(* PLC project Traffic control simulator, CODESYS CODESYS V3.5 SP16, author Toni Kucic *)
(* stored: creationDateTime 2021-03-25T19:26:30.1030266, version 1.0, modificationDateTime 2021-03-25T19:26:13.0193121, organization TK Automation *)
(* Traffic control is often used a simple introduction into sequencing when programming PLCs. As a part of my portfolio I have written a simple timing controller and a simulator for two crossroads that are one way streets with pedestrians going in all directions. The project is meant for begginers and for educational purposes. It is published under MIT license. Written in CODESYS 3.5 and in structured text language. *)

TYPE SpriteDef_typ : STRUCT
  x : INT;  (* Initial position of the sprite *)
  y : INT;  (* Initial position of the sprite *)
  speed : INT;  (* Initial speed of the sprite *)
  width : INT;  (* Sprites width *)
  height : INT;  (* Sprites height *)
  screenWidth : INT;  (* Screen width *)
  screenHeight : INT;  (* Screen height *)
END_STRUCT;
END_TYPE

TYPE trafficLightCars : STRUCT
  RedLamp : BOOL;  (* TRUE: Red lamp is on *)
  YellowLamp : BOOL;  (* TRUE: Yellow lamp is on *)
  GreenLamp : BOOL;  (* TRUE: Green lamp is on *)
END_STRUCT;
END_TYPE

TYPE trafficLightPed : STRUCT
  RedLight : BOOL;  (* TRUE: Red lamp is on *)
  GreenLight : BOOL;  (* TRUE: Green lamp is on *)
  TimeToSequenceChange : UINT;  (* Time in seconds until next light change *)
END_STRUCT;
END_TYPE

FUNCTION isSpriteColliding : BOOL
  VAR_INPUT
    sprite1 : Sprite;  (* Sprite 1 function block *)
    sprite2 : Sprite;  (* Sprite 2 function block *)
  END_VAR

            (*Calculate if these two sprites are overlapping*)
IF sprite1.actX < (sprite2.actX + sprite2.init.width) AND
   (sprite1.actX + sprite1.init.width) > sprite2.actX AND
   sprite1.actY < (sprite2.actY + sprite2.init.height) AND
  ( sprite1.init.height + sprite1.actY) > sprite2.actY THEN
   isSpriteColliding := TRUE;
ELSE
	isSpriteColliding := FALSE;
END_IF
          
END_FUNCTION

FUNCTION_BLOCK Sprite
  VAR_INPUT
    init : SpriteDef_typ;  (* Sprite initialization pars *)
    goTo : ARRAY[0..1] OF INT;  (* Sprite moves to x,y destination *)
    moveX : INT;  (* Moves the sprite by given ammount on the X axis *)
    moveY : INT;  (* Moves the sprite by given ammount on the Y axis *)
  END_VAR
  VAR_OUTPUT
    x : INT;  (* X position of the sprite *)
    y : INT;  (* Y position of the sprite *)
    atDestination : BOOL;  (* Flag to say it has arrived at its destination *)
    actX : INT;  (* Actual position on the screen, X axis *)
    actY : INT;  (* Actual position on the screen, Y axis *)
  END_VAR
  VAR
    vInit : BOOL := TRUE;  (* Initialization flag *)
    vSpriteDef : SpriteDef_typ;  (* Used sprite definition *)
    vActualX : INT;  (* Actual position on the screen, X axis *)
    vActualY : INT;  (* Actual position on the screen, Y axis *)
  END_VAR

            (*Initialize sprite on first scan*)
IF vInit THEN
	vSpriteDef := init;
	vInit := FALSE;
END_IF

(* Actual moving of the coordinates *)
vSpriteDef.x := vSpriteDef.x + moveX;
vSpriteDef.y := vSpriteDef.y + moveY;

(* Reseting the position if sprite goes off screen *)
(* If moving left to right *)
IF vSpriteDef.x > vSpriteDef.screenWidth THEN
	vSpriteDef.x := -vSpriteDef.width;
(* If moving right to left *)
ELSIF vSpriteDef.x < -vSpriteDef.width THEN
	vSpriteDef.x := vSpriteDef.screenWidth;	
END_IF
(* If moving from up, down *)
IF vSpriteDef.y > vSpriteDef.screenHeight THEN
	vSpriteDef.y := -vSpriteDef.height;
(* If moving from down, up *)
ELSIF vSpriteDef.y < -vSpriteDef.height THEN
	vSpriteDef.y := vSpriteDef.screenHeight;	
END_IF

(*x, y will be used to connect to absoulte movements of the graphic element*)
x := vSpriteDef.x - init.x;
y := vSpriteDef.y - init.y;

(*ActX and ActY will be used in the logic for e.g. object collision detection*)
actX := vSpriteDef.x;
actY := vSpriteDef.y;
          
END_FUNCTION_BLOCK

PROGRAM simulator
  VAR
    carC1HR : Sprite := (init := (screenHeight := 720, screenWidth := 1980, height := 80, width := 200, x := 568, y := 264));  (* Sprite controling car C1HR *)
    carC1HL : Sprite := (init := (screenHeight := 720, screenWidth := 1980, height := 80, width := 200, x := -50, y := 370));  (* Sprite controling car C1HL *)
    carC1VU : Sprite := (init := (screenHeight := 720, screenWidth := 1980, height := 200, width := 80, x := 270, y := -50));  (* Sprite controling car C1VU *)
    carC1VD : Sprite := (init := (screenHeight := 720, screenWidth := 1980, height := 200, width := 80, x := 372, y := 565));  (* Sprite controling car C1VD *)
    carC2VU : Sprite := (init := (screenHeight := 720, screenWidth := 1980, height := 200, width := 80, x := 1528, y := -50));  (* Sprite controling car C2VU *)
    carC2VD : Sprite := (init := (screenHeight := 720, screenWidth := 1980, height := 200, width := 80, x := 1631, y := 580));  (* Sprite controling car C2VD *)
    pedC1VU : Sprite := (init := (screenHeight := 720, screenWidth := 1980, height := 50, width := 50, x := 171, y := 7));  (* Sprite controling pedestrian C1VU *)
    pedC1VD : Sprite := (init := (screenHeight := 720, screenWidth := 1980, height := 50, width := 50, x := 486, y := 657));  (* Sprite controling pedestrian C1VD *)
    pedC2VU : Sprite := (init := (screenHeight := 720, screenWidth := 1980, height := 50, width := 50, x := 1427, y := 2));  (* Sprite controling pedestrian C2VU *)
    pedC2VD : Sprite := (init := (screenHeight := 720, screenWidth := 1980, height := 50, width := 50, x := 1742, y := 654));  (* Sprite controling pedestrian C2VD *)
    pedC1HL : Sprite := (init := (screenHeight := 720, screenWidth := 1980, height := 50, width := 50, x := 9, y := 491));  (* Sprite controling pedestrian C1HL *)
    pedC2HR : Sprite := (init := (screenHeight := 720, screenWidth := 1980, height := 50, width := 50, x := 1916, y := 174));  (* Sprite controling pedestrian C1HR *)
    Cross1CarU : trafficLightCars;  (* Car traffic light - Crossroad 1 - Cars going up to down *)
    Cross1CarD : trafficLightCars;  (* Car traffic light - Crossroad 1 - Cars going down to up *)
    Cross1CarL : trafficLightCars;  (* Car traffic light - Crossroad 1 - Cars going left to right *)
    Cross1CarR : trafficLightCars;  (* Car traffic light - Crossroad 1 - Cars going right to left *)
    Cross2CarU : trafficLightCars;  (* Car light - Crossroad 2 - Cars going up to down *)
    Cross2CarD : trafficLightCars;  (* Car light - Crossroad 2 - Cars going down to up *)
    Cross2CarL : trafficLightCars;  (* Car light - Crossroad 2 - Cars going left to right *)
    Cross2CarR : trafficLightCars;  (* Car light - Crossroad 2 - Cars going right to left *)
    Cross1PedLUD : trafficLightPed;  (* Pedestrian light - Crossroad 1 - Pedestrians going up to down on left side *)
    Cross1PedLDU : trafficLightPed;  (* Pedestrian light - Crossroad 1 - Pedestrians going down to up on left side *)
    Cross1PedRUD : trafficLightPed;  (* Pedestrian light - Crossroad 1 - Pedestrians going up to down on right side *)
    Cross1PedRDU : trafficLightPed;  (* Pedestrian light - Crossroad 1 - Pedestrians going down to up on right side *)
    Cross1PedULR : trafficLightPed;  (* Pedestrian light - Crossroad 1 - Pedestrians going left to right on upper side *)
    Cross1PedURL : trafficLightPed;  (* Pedestrian light - Crossroad 1 - Pedestrians going right to left on upper side *)
    Cross1PedDLR : trafficLightPed;  (* Pedestrian light - Crossroad 1 - Pedestrians going left to right on lower side *)
    Cross1PedDRL : trafficLightPed;  (* Pedestrian light - Crossroad 1 - Pedestrians going right to left on lower side *)
    Cross2PedLUD : trafficLightPed;  (* Pedestrian light - Crossroad 2 - Pedestrians going up to down on left side *)
    Cross2PedLDU : trafficLightPed;  (* Pedestrian light - Crossroad 2 - Pedestrians going down to up on left side *)
    Cross2PedRUD : trafficLightPed;  (* Pedestrian light - Crossroad 2 - Pedestrians going up to down on right side *)
    Cross2PedRDU : trafficLightPed;  (* Pedestrian light - Crossroad 2 - Pedestrians going down to up on right side *)
    Cross2PedULR : trafficLightPed;  (* Pedestrian light - Crossroad 2 - Pedestrians going left to right on upper side *)
    Cross2PedURL : trafficLightPed;  (* Pedestrian light - Crossroad 2 - Pedestrians going right to left on upper side *)
    Cross2PedDLR : trafficLightPed;  (* Pedestrian light - Crossroad 2 - Pedestrians going left to right on lower side *)
    Cross2PedDRL : trafficLightPed;  (* Pedestrian light - Crossroad 2 - Pedestrians going right to left on lower side *)
    vCollision : BOOL;  (* Collission has occured *)
    vDangerousCombination : BOOL;  (* Dangerous combination of lights has been detected *)
    vPoliceControl : BOOL;  (* Police control activated *)
    vCrashFlagX : INT := -200;  (* If collission is detected, holds position of collission x axis *)
    vCrashFlagY : INT := -200;  (* If collission is detected, holds position of collission y axis *)
    Blinker : BLINK;  (* Code that blinks a variable *)
    vFaultReason : STRING(255);  (* If collission or dangerous combination detected, holds more information where it has occured *)
  END_VAR

                    MOVE_CARS();
MOVE_PEDESTRIANS();

(*Blink yellow signal if the police is under control*)
IF vPoliceControl THEN
	UPDATE_OBJECTS();
	BLINK_YELLOW_SIGNAL();
(*Freeze situation if a collission or dangerous situation has occured*)
ELSIF vCollision OR vDangerousCombination THEN
	BLINK_DANGER_SIGNAL();
ELSE
	(*Everything is fine so move objects and let the main control the lights*)
	UPDATE_OBJECTS();
	CONTROL_LIGHTS();
	vFaultReason := '';
END_IF
FAULT_MONITOR();
gIO.PoliceModeActivated := vPoliceControl;
Blinker(ENABLE:=TRUE, TIMELOW:=T#1S, TIMEHIGH:=T#1S);



                  

ACTION CHECK_COLLISSIONS:
                        (*Check for collisions between each car with another car and pedestrian*)
vCollision := FALSE;

(*Collission car -> car*)
IF isSpriteColliding(carC1HR, carC1HL) THEN
	vCollision := TRUE;
	vCrashFlagX := carC1HR.actX;
	vCrashFlagY := carC1HL.actY;
	vFaultReason := 'COLLISSION AT CAR C1HR AND CAR C1HL';
END_IF
IF isSpriteColliding(carC1HR, carC1VU) THEN
	vCollision := TRUE;
	vCrashFlagX := carC1HR.actX;
	vCrashFlagY := carC1VU.actY;
	vFaultReason := 'COLLISSION AT CAR C1HR AND CAR C1VU';
END_IF
IF isSpriteColliding(carC1HR, carC1VD) THEN
	vCollision := TRUE;
	vCrashFlagX := carC1HR.actX;
	vCrashFlagY := carC1VD.actY;
	vFaultReason := 'COLLISSION AT CAR C1HR AND CAR C1VD';
END_IF
IF isSpriteColliding(carC1HR, carC2VD) THEN
	vCollision := TRUE;
	vCrashFlagX := carC1HR.actX;
	vCrashFlagY := carC2VD.actY;
	vFaultReason := 'COLLISSION AT CAR C1HR AND CAR C2VD';
END_IF
IF isSpriteColliding(carC1HR, carC2VU) THEN
	vCollision := TRUE;
	vCrashFlagX := carC1HR.actX;
	vCrashFlagY := carC2VU.actY;
	vFaultReason := 'COLLISSION AT CAR C1HR AND CAR C2VU';
END_IF
IF isSpriteColliding(carC1HL, carC1VU) THEN
	vCollision := TRUE;
	vCrashFlagX := carC1HL.actX;
	vCrashFlagY := carC1VU.actY;
	vFaultReason := 'COLLISSION AT CAR C1HL AND CAR C1VU';
END_IF
IF isSpriteColliding(carC1HL, carC1VD) THEN
	vCollision := TRUE;
	vCrashFlagX := carC1HL.actX;
	vCrashFlagY := carC1VD.actY;
	vFaultReason := 'COLLISSION AT CAR C1HL AND CAR C1VD';
END_IF
IF isSpriteColliding(carC1HL, carC2VU) THEN
	vCollision := TRUE;
	vCrashFlagX := carC1HL.actX;
	vCrashFlagY := carC2VU.actY;
	vFaultReason := 'COLLISSION AT CAR C1HL AND CAR C2VU';
END_IF
IF isSpriteColliding(carC1HL, carC2VD) THEN
	vCollision := TRUE;
	vCrashFlagX := carC1HL.actX;
	vCrashFlagY := carC2VD.actY;
	vFaultReason := 'COLLISSION AT CAR C1HL AND CAR C2VD';
END_IF
IF isSpriteColliding(carC1VU, carC1VD) THEN
	vCollision := TRUE;
	vCrashFlagX := carC1VU.actX;
	vCrashFlagY := carC1VD.actY;
	vFaultReason := 'COLLISSION AT CAR C1VU AND CAR C1VD';
END_IF
IF isSpriteColliding(carC1VU, carC2VD) THEN
	vCollision := TRUE;
	vCrashFlagX := carC1VU.actX;
	vCrashFlagY := carC2VD.actY;
	vFaultReason := 'COLLISSION AT CAR C1VU AND CAR C2VD';
END_IF
IF isSpriteColliding(carC1VU, carC2VU) THEN
	vCollision := TRUE;
	vCrashFlagX := carC1VU.actX;
	vCrashFlagY := carC2VU.actY;
	vFaultReason := 'COLLISSION AT CAR C1VU AND CAR C2VU';
END_IF
IF isSpriteColliding(carC1VD, carC2VD) THEN
	vCollision := TRUE;
	vCrashFlagX := carC1VD.actX;
	vCrashFlagY := carC2VD.actY;
	vFaultReason := 'COLLISSION AT CAR C1VD AND CAR C2VD';
END_IF
IF isSpriteColliding(carC1VD, carC2VU) THEN
	vCollision := TRUE; 
	vCrashFlagX := carC1VD.actX;
	vCrashFlagY := carC2VU.actY;
	vFaultReason := 'COLLISSION AT CAR C1VD AND CAR C2VU';
END_IF
IF isSpriteColliding(carC2VD, carC2VU) THEN
	vCollision := TRUE; 
	vCrashFlagX := carC2VD.actX;
	vCrashFlagY := carC2VU.actY;
	vFaultReason := 'COLLISSION AT CAR C2VD AND CAR C2VU';
END_IF

(*Check collission car -> pedestrian*)
IF isSpriteColliding(carC1HR, pedC1HL) THEN
	vCollision := TRUE;
	vCrashFlagX := carC1HR.actX;
	vCrashFlagY := pedC1HL.actY;
	vFaultReason := 'COLLISSION AT CAR C1HR AND PEDESTRIAN C1HL';
END_IF
IF isSpriteColliding(carC1HR, pedC1VU) THEN
	vCollision := TRUE;
	vCrashFlagX := carC1HR.actX;
	vCrashFlagY := pedC1VU.actY;
	vFaultReason := 'COLLISSION AT CAR C1HR AND PEDESTRIAN C1VU';
END_IF
IF isSpriteColliding(carC1HR, pedC1VD) THEN
	vCollision := TRUE;
	vCrashFlagX := carC1HR.actX;
	vCrashFlagY := pedC1VD.actY;
	vFaultReason := 'COLLISSION AT CAR C1HR AND PEDESTRIAN C1VD';
END_IF
IF isSpriteColliding(carC1HR, pedC2VU) THEN
	vCollision := TRUE;
	vCrashFlagX := carC1HR.actX;
	vCrashFlagY := pedC2VU.actY;
	vFaultReason := 'COLLISSION AT CAR C1HR AND PEDESTRIAN C2VU';
END_IF
IF isSpriteColliding(carC1HR, pedC2VD) THEN
	vCollision := TRUE;
	vCrashFlagX := carC1HR.actX;
	vCrashFlagY := pedC2VD.actY;
	vFaultReason := 'COLLISSION AT CAR C1HR AND PEDESTRIAN C2VD';
END_IF
IF isSpriteColliding(carC1HR, pedC2HR) THEN
	vCollision := TRUE;
	vCrashFlagX := carC1HR.actX;
	vCrashFlagY := pedC2HR.actY;
	vFaultReason := 'COLLISSION AT CAR C1HR AND PEDESTRIAN C2HR';
END_IF


IF isSpriteColliding(carC1HL, pedC1HL) THEN
	vCollision := TRUE;
	vCrashFlagX := carC1HL.actX;
	vCrashFlagY := pedC1HL.actY;
	vFaultReason := 'COLLISSION AT CAR C1HL AND PEDESTRIAN C1HL';
END_IF
IF isSpriteColliding(carC1HL, pedC1VU) THEN
	vCollision := TRUE;
	vCrashFlagX := carC1HL.actX;
	vCrashFlagY := pedC1VU.actY;
	vFaultReason := 'COLLISSION AT CAR C1HL AND PEDESTRIAN C1VU';
END_IF
IF isSpriteColliding(carC1HL, pedC1VD) THEN
	vCollision := TRUE;
	vCrashFlagX := carC1HL.actX;
	vCrashFlagY := pedC1VD.actY;
	vFaultReason := 'COLLISSION AT CAR C1HL AND PEDESTRIAN C1VD';
END_IF
IF isSpriteColliding(carC1HL, pedC2VU) THEN
	vCollision := TRUE;
	vCrashFlagX := carC1HL.actX;
	vCrashFlagY := pedC2VU.actY;
	vFaultReason := 'COLLISSION AT CAR C1HL AND PEDESTRIAN C2VU';
END_IF
IF isSpriteColliding(carC1HL, pedC2VD) THEN
	vCollision := TRUE;
	vCrashFlagX := carC1HL.actX;
	vCrashFlagY := pedC2VD.actY;
	vFaultReason := 'COLLISSION AT CAR C1HL AND PEDESTRIAN C2VD';
END_IF
IF isSpriteColliding(carC1HL, pedC2HR) THEN
	vCollision := TRUE;
	vCrashFlagX := carC1HL.actX;
	vCrashFlagY := pedC2HR.actY;
	vFaultReason := 'COLLISSION AT CAR C1HL AND PEDESTRIAN C2HR';
END_IF


IF isSpriteColliding(carC1VU, pedC1HL) THEN
	vCollision := TRUE;
	vCrashFlagX := carC1VU.actX;
	vCrashFlagY := pedC1HL.actY;
	vFaultReason := 'COLLISSION AT CAR C1VU AND PEDESTRIAN C1HL';
END_IF
IF isSpriteColliding(carC1VU, pedC1VU) THEN
	vCollision := TRUE;
	vCrashFlagX := carC1VU.actX;
	vCrashFlagY := pedC1VU.actY;
	vFaultReason := 'COLLISSION AT CAR C1VU AND PEDESTRIAN C1VU';
END_IF
IF isSpriteColliding(carC1VU, pedC1VD) THEN
	vCollision := TRUE;
	vCrashFlagX := carC1VU.actX;
	vCrashFlagY := pedC1VD.actY;
	vFaultReason := 'COLLISSION AT CAR C1VU AND PEDESTRIAN C1VD';
END_IF
IF isSpriteColliding(carC1VU, pedC2VU) THEN
	vCollision := TRUE;
	vCrashFlagX := carC1VU.actX;
	vCrashFlagY := pedC2VU.actY;
	vFaultReason := 'COLLISSION AT CAR C1VU AND PEDESTRIAN C2VU';
END_IF
IF isSpriteColliding(carC1VU, pedC2VD) THEN
	vCollision := TRUE;
	vCrashFlagX := carC1VU.actX;
	vCrashFlagY := pedC2VD.actY;
	vFaultReason := 'COLLISSION AT CAR C1VU AND PEDESTRIAN C2VD';
END_IF
IF isSpriteColliding(carC1VU, pedC2HR) THEN
	vCollision := TRUE;
	vCrashFlagX := carC1VU.actX;
	vCrashFlagY := pedC2HR.actY;
	vFaultReason := 'COLLISSION AT CAR C1VU AND PEDESTRIAN C2HR';
END_IF


IF isSpriteColliding(carC1VD, pedC1HL) THEN
	vCollision := TRUE;
	vCrashFlagX := carC1VD.actX;
	vCrashFlagY := pedC1HL.actY;
	vFaultReason := 'COLLISSION AT CAR C1VD AND PEDESTRIAN C1HL';
END_IF
IF isSpriteColliding(carC1VD, pedC1VU) THEN
	vCollision := TRUE;
	vCrashFlagX := carC1VD.actX;
	vCrashFlagY := pedC1VU.actY;
	vFaultReason := 'COLLISSION AT CAR C1VD AND PEDESTRIAN C1VU';
END_IF
IF isSpriteColliding(carC1VD, pedC1VD) THEN
	vCollision := TRUE;
	vCrashFlagX := carC1VD.actX;
	vCrashFlagY := pedC1VD.actY;
	vFaultReason := 'COLLISSION AT CAR C1VD AND PEDESTRIAN C1VD';
END_IF
IF isSpriteColliding(carC1VD, pedC2VU) THEN
	vCollision := TRUE;
	vCrashFlagX := carC1VD.actX;
	vCrashFlagY := pedC2VU.actY;
	vFaultReason := 'COLLISSION AT CAR C1VD AND PEDESTRIAN C2VU';
END_IF
IF isSpriteColliding(carC1VD, pedC2VD) THEN
	vCollision := TRUE;
	vCrashFlagX := carC1VD.actX;
	vCrashFlagY := pedC2VD.actY;
	vFaultReason := 'COLLISSION AT CAR C1VD AND PEDESTRIAN C2VD';
END_IF
IF isSpriteColliding(carC1VD, pedC2HR) THEN
	vCollision := TRUE;
	vCrashFlagX := carC1VD.actX;
	vCrashFlagY := pedC2HR.actY;
	vFaultReason := 'COLLISSION AT CAR C1VD AND PEDESTRIAN C2HR';
END_IF


IF isSpriteColliding(carC2VU, pedC1HL) THEN
	vCollision := TRUE;
	vCrashFlagX := carC2VU.actX;
	vCrashFlagY := pedC1HL.actY;
	vFaultReason := 'COLLISSION AT CAR C2VU AND PEDESTRIAN C1HL';
END_IF
IF isSpriteColliding(carC2VU, pedC1VU) THEN
	vCollision := TRUE;
	vCrashFlagX := carC2VU.actX;
	vCrashFlagY := pedC1VU.actY;
	vFaultReason := 'COLLISSION AT CAR C2VU AND PEDESTRIAN C1VU';
END_IF
IF isSpriteColliding(carC2VU, pedC1VD) THEN
	vCollision := TRUE;
	vCrashFlagX := carC2VU.actX;
	vCrashFlagY := pedC1VD.actY;
	vFaultReason := 'COLLISSION AT CAR C2VU AND PEDESTRIAN C1VD';
END_IF
IF isSpriteColliding(carC2VU, pedC2VU) THEN
	vCollision := TRUE;
	vCrashFlagX := carC2VU.actX;
	vCrashFlagY := pedC2VU.actY;
	vFaultReason := 'COLLISSION AT CAR C2VU AND PEDESTRIAN C2VU';
END_IF
IF isSpriteColliding(carC2VU, pedC2VD) THEN
	vCollision := TRUE;
	vCrashFlagX := carC2VU.actX;
	vCrashFlagY := pedC2VD.actY;
	vFaultReason := 'COLLISSION AT CAR C2VU AND PEDESTRIAN C2VD';
END_IF
IF isSpriteColliding(carC2VU, pedC2HR) THEN
	vCollision := TRUE;
	vCrashFlagX := carC2VU.actX;
	vCrashFlagY := pedC2HR.actY;
	vFaultReason := 'COLLISSION AT CAR C2VU AND PEDESTRIAN C2HR';
END_IF


IF isSpriteColliding(carC2VD, pedC1HL) THEN
	vCollision := TRUE;
	vCrashFlagX := carC2VD.actX;
	vCrashFlagY := pedC1HL.actY;
	vFaultReason := 'COLLISSION AT CAR C2VD AND PEDESTRIAN C1HL';
END_IF
IF isSpriteColliding(carC2VD, pedC1VU) THEN
	vCollision := TRUE;
	vCrashFlagX := carC2VD.actX;
	vCrashFlagY := pedC1VU.actY;
	vFaultReason := 'COLLISSION AT CAR C2VD AND PEDESTRIAN pedC1VU';
END_IF
IF isSpriteColliding(carC2VD, pedC1VD) THEN
	vCollision := TRUE;
	vCrashFlagX := carC2VD.actX;
	vCrashFlagY := pedC1VD.actY;
	vFaultReason := 'COLLISSION AT CAR C2VD AND PEDESTRIAN C1VD';
END_IF
IF isSpriteColliding(carC2VD, pedC2VU) THEN
	vCollision := TRUE;
	vCrashFlagX := carC2VD.actX;
	vCrashFlagY := pedC2VU.actY;
	vFaultReason := 'COLLISSION AT CAR C2VD AND PEDESTRIAN C2VU';
END_IF
IF isSpriteColliding(carC2VD, pedC2VD) THEN
	vCollision := TRUE;
	vCrashFlagX := carC2VD.actX;
	vCrashFlagY := pedC2VD.actY;
	vFaultReason := 'COLLISSION AT CAR C2VD AND PEDESTRIAN C2VD';
END_IF
IF isSpriteColliding(carC2VD, pedC2HR) THEN
	vCollision := TRUE;
	vCrashFlagX := carC2VD.actX;
	vCrashFlagY := pedC2HR.actY;
	vFaultReason := 'COLLISSION AT CAR C2VD AND PEDESTRIAN C2HR';
END_IF

(*Hide the crash flag if there is no collission*)
IF NOT vCollision THEN
	vCrashFlagX := -200;
	vCrashFlagY := -200;
END_IF

                      
END_ACTION

ACTION MOVE_CARS:
                        (*Car C1 HL. Moves from left to right, stops at the crossroads and moves if only green is lit*)
IF carC1HL.actX = -49 THEN
	IF (Cross1CarL.GreenLamp AND NOT (Cross1CarL.RedLamp OR Cross1CarL.YellowLamp)) THEN
		carC1HL.moveX := 1;
	ELSE
		carC1HL.moveX := 0;
	END_IF
ELSIF carC1HL.actX = 1211 THEN
	IF (Cross2CarL.GreenLamp AND NOT (Cross2CarL.RedLamp OR Cross2CarL.YellowLamp)) THEN
		carC1HL.moveX := 1;
	ELSE
		carC1HL.moveX := 0;
	END_IF
ELSE
	carC1HL.moveX := 1;
END_IF

(*Car C1 HR. Moves from right to left, stops at the crossroads and moves if only green is lit*)
IF carC1HR.actX = 567 THEN
	IF (Cross1CarR.GreenLamp AND NOT (Cross1CarR.RedLamp OR Cross1CarR.YellowLamp)) THEN
		carC1HR.moveX := -1;
	ELSE
		carC1HR.moveX := 0;
	END_IF
ELSIF carC1HR.actX = 1829 THEN
	IF (Cross2CarR.GreenLamp AND NOT (Cross2CarR.RedLamp OR Cross2CarR.YellowLamp)) THEN
		carC1HR.moveX := -1;
	ELSE
		carC1HR.moveX := 0;
	END_IF
ELSE
	carC1HR.moveX := -1;
END_IF
(*Car C1 VU. Moves from up to down, stops at the crossroads and moves if only green is lit*)
IF carC1VU.actY = -49 THEN
	IF (Cross1CarU.GreenLamp AND NOT (Cross1CarU.RedLamp OR Cross1CarU.YellowLamp)) THEN
		carC1VU.moveY := 1;
	ELSE
		carC1VU.moveY := 0;
	END_IF
ELSE
	carC1VU.moveY := 1;
END_IF
(*Car C2 VU. Moves from up to down, stops at the crossroads and moves if only green is lit*)
IF carC2VU.actY = -49 THEN
	IF (Cross2CarU.GreenLamp AND NOT (Cross2CarU.RedLamp OR Cross2CarU.YellowLamp)) THEN
		carC2VU.moveY := 1;
	ELSE
		carC2VU.moveY := 0;
	END_IF
ELSE
	carC2VU.moveY := 1;
END_IF
(*Car C1 VD. Moves from down to up, stops at the crossroads and moves if only green is lit*)
IF carC1VD.actY = 564 THEN
	IF (Cross1CarD.GreenLamp AND NOT (Cross1CarD.RedLamp OR Cross1CarD.YellowLamp)) THEN
		carC1VD.moveY := -1;
	ELSE
		carC1VD.moveY := 0;
	END_IF
ELSE
	carC1VD.moveY := -1;
END_IF
(*Car C2 VD. Moves from down to up, stops at the crossroads and moves if only green is lit*)
IF carC2VD.actY = 564 THEN
	IF (Cross2CarD.GreenLamp AND NOT (Cross2CarD.RedLamp OR Cross2CarD.YellowLamp)) THEN
		carC2VD.moveY := -1;
	ELSE
		carC2VD.moveY := 0;
	END_IF
ELSE
	carC2VD.moveY := -1;
END_IF
                      
END_ACTION

ACTION MOVE_PEDESTRIANS:
                        (*Pedestrian C1 VU. Moves from up to down, stops at the crossroads and moves if only green is lit*)
IF pedC1VU.actY = 180 THEN
	IF Cross1PedLUD.GreenLight AND NOT Cross1PedLUD.RedLight THEN
		pedC1VU.moveY := 1;
	ELSE
		pedC1VU.moveY := 0;
	END_IF
ELSE
	pedC1VU.moveY := 1;
END_IF
(*Pedestrian C2 VU. Moves from up to down, stops at the crossroads and moves if only green is lit*)
IF pedC2VU.actY = 180 THEN
	IF Cross2PedLUD.GreenLight AND NOT Cross2PedLUD.RedLight THEN
		pedC2VU.moveY := 1;
	ELSE
		pedC2VU.moveY := 0;
	END_IF
ELSE
	pedC2VU.moveY := 1;
END_IF
(*Pedestrian C1 VD. Moves from down to up, stops at the crossroads and moves if only green is lit*)
IF pedC1VD.actY = 480 THEN
	IF Cross1PedLDU.GreenLight AND NOT Cross1PedLDU.RedLight THEN
		pedC1VD.moveY := -1;
	ELSE
		pedC1VD.moveY := 0;
	END_IF
ELSE
	pedC1VD.moveY := -1;
END_IF
(*Pedestrian C1 VD. Moves from down to up, stops at the crossroads and moves if only green is lit*)
IF pedC2VD.actY = 480 THEN
	IF Cross2PedLDU.GreenLight AND NOT Cross2PedLDU.RedLight THEN
		pedC2VD.moveY := -1;
	ELSE
		pedC2VD.moveY := 0;
	END_IF
ELSE
	pedC2VD.moveY := -1;
END_IF
(*Pedestrian C1 HL. Moves from left to right, stops at the crossroads and moves if only green is lit*)
IF pedC1HL.actX = 190 THEN
	IF Cross1PedDLR.GreenLight AND NOT Cross1PedDLR.RedLight THEN
		pedC1HL.moveX := 1;
	ELSE
		pedC1HL.moveX := 0;
	END_IF
ELSIF pedC1HL.actX = 1450 THEN
	IF Cross2PedDLR.GreenLight AND NOT Cross2PedDLR.RedLight THEN
		pedC1HL.moveX := 1;
	ELSE
		pedC1HL.moveX := 0;
	END_IF
ELSE
	pedC1HL.moveX := 1;
END_IF
(*Pedestrian C1 HR. Moves from right to left, stops at the crossroads and moves if only green is lit*)
IF pedC2HR.actX = 1740 THEN
	IF Cross2PedURL.GreenLight AND NOT Cross2PedURL.RedLight THEN
		pedC2HR.moveX := -1;
	ELSE
		pedC2HR.moveX := 0;
	END_IF
ELSIF pedC2HR.actX = 480 THEN
	IF Cross1PedURL.GreenLight AND NOT Cross1PedURL.RedLight THEN
		pedC2HR.moveX := -1;
	ELSE
		pedC2HR.moveX := 0;
	END_IF
ELSE
	pedC2HR.moveX := -1;
END_IF
                      
END_ACTION

ACTION UPDATE_OBJECTS:
                        // Update sprites
carC1HR();
carC1HL();
carC1VD();
carC1VU();
carC2VD();
carC2VU();
pedC1VU();
pedC1VD();
pedC2VU();
pedC2VD();
pedC1HL();
pedC2HR();
                      
END_ACTION

ACTION CONTROL_LIGHTS:
                        Cross1CarU := gIO.Cross1CarU;
Cross1CarD := gIO.Cross1CarD;
Cross1CarL := gIO.Cross1CarL;
Cross1CarR := gIO.Cross1CarR;

Cross2CarU := gIO.Cross2CarU;
Cross2CarD := gIO.Cross2CarD;
Cross2CarL := gIO.Cross2CarL;
Cross2CarR := gIO.Cross2CarR;

Cross1PedLUD := gIO.Cross1PedLUD;
Cross1PedLDU := gIO.Cross1PedLDU;
Cross1PedRUD := gIO.Cross1PedRUD;
Cross1PedRDU := gIO.Cross1PedRDU;

Cross1PedULR := gIO.Cross1PedULR;
Cross1PedURL := gIO.Cross1PedURL;
Cross1PedDLR := gIO.Cross1PedDLR;
Cross1PedDRL := gIO.Cross1PedDRL;

Cross2PedLUD := gIO.Cross2PedLUD;
Cross2PedLDU := gIO.Cross2PedLDU;
Cross2PedRUD := gIO.Cross2PedRUD;
Cross2PedRDU := gIO.Cross2PedRDU;

Cross2PedULR := gIO.Cross2PedULR;
Cross2PedURL := gIO.Cross2PedURL;
Cross2PedDLR := gIO.Cross2PedDLR;
Cross2PedDRL := gIO.Cross2PedDRL;
                      
END_ACTION

ACTION FAULT_MONITOR:
                        (*Checks if dangerous situations occur, horizontal wave and vertical wave green at the same time*)
vDangerousCombination := FALSE;
(*Green vertical and horizontal pedestrians green*)
IF Cross1CarU.GreenLamp AND (Cross1PedULR.GreenLight OR Cross1PedURL.GreenLight) THEN
	vDangerousCombination := TRUE;
	vFaultReason := 'DANGEROUS COMBINATION AT CROSS1 -> VERTICAL CARS AND HORIZONTAL PEDESTRIANS GREEN AT THE SAME TIME';
END_IF
IF Cross2CarU.GreenLamp AND (Cross2PedULR.GreenLight OR Cross2PedURL.GreenLight) THEN
	vDangerousCombination := TRUE;
	vFaultReason := 'DANGEROUS COMBINATION AT CROSS2 -> VERTICAL CARS AND HORIZONTAL PEDESTRIANS GREEN AT THE SAME TIME';
END_IF
IF Cross1CarD.GreenLamp AND (Cross1PedDLR.GreenLight OR Cross1PedDRL.GreenLight) THEN
	vDangerousCombination := TRUE;
	vFaultReason := 'DANGEROUS COMBINATION AT CROSS1 -> VERTICAL CARS AND HORIZONTAL PEDESTRIANS GREEN AT THE SAME TIME';
END_IF
IF Cross2CarD.GreenLamp AND (Cross2PedDLR.GreenLight OR Cross2PedDRL.GreenLight) THEN
	vDangerousCombination := TRUE;
	vFaultReason := 'DANGEROUS COMBINATION AT CROSS2 -> VERTICAL CARS AND HORIZONTAL PEDESTRIANS GREEN AT THE SAME TIME';
END_IF

(*Green horizontal and vertical pedestrians green*)
IF Cross1CarL.GreenLamp AND (Cross1PedLUD.GreenLight OR Cross1PedLDU.GreenLight) THEN
	vDangerousCombination := TRUE;
	vFaultReason := 'DANGEROUS COMBINATION AT CROSS1 -> HORIZONTAL CARS AND VERTICAL PEDESTRIANS GREEN AT THE SAME TIME';
END_IF
IF Cross1CarR.GreenLamp AND (Cross1PedRUD.GreenLight OR Cross1PedRDU.GreenLight) THEN
	vDangerousCombination := TRUE;
	vFaultReason := 'DANGEROUS COMBINATION AT CROSS1 -> HORIZONTAL CARS AND VERTICAL PEDESTRIANS GREEN AT THE SAME TIME';
END_IF
IF Cross2CarL.GreenLamp AND (Cross2PedLUD.GreenLight OR Cross2PedLDU.GreenLight) THEN
	vDangerousCombination := TRUE;
	vFaultReason := 'DANGEROUS COMBINATION AT CROSS2 -> HORIZONTAL CARS AND VERTICAL PEDESTRIANS GREEN AT THE SAME TIME';
END_IF
IF Cross2CarR.GreenLamp AND (Cross2PedRUD.GreenLight OR Cross2PedRDU.GreenLight) THEN
	vDangerousCombination := TRUE;
	vFaultReason := 'DANGEROUS COMBINATION AT CROSS2 -> HORIZONTAL CARS AND VERTICAL PEDESTRIANS GREEN AT THE SAME TIME';
END_IF

(*Checks if there was a collission with car-car and ped - car*)
CHECK_COLLISSIONS();
                      
END_ACTION

ACTION BLINK_DANGER_SIGNAL:
                        Cross1CarU.GreenLamp := FALSE;
Cross1CarU.YellowLamp := FALSE;
Cross1CarU.RedLamp := Blinker.OUT;

Cross1CarD := Cross1CarU;
Cross1CarL := Cross1CarU;
Cross1CarR := Cross1CarU;

Cross2CarU := Cross1CarU;
Cross2CarD := Cross1CarU;
Cross2CarL := Cross1CarU;
Cross2CarR := Cross1CarU;

Cross1PedLUD.GreenLight := FALSE;
Cross1PedLUD.RedLight := Blinker.OUT;
Cross1PedLUD.TimeToSequenceChange := 0;

Cross1PedLDU := Cross1PedLUD;
Cross1PedRUD := Cross1PedLUD;
Cross1PedRDU := Cross1PedLUD;

Cross1PedULR := Cross1PedLUD;
Cross1PedURL := Cross1PedLUD;
Cross1PedDLR := Cross1PedLUD;
Cross1PedDRL := Cross1PedLUD;

Cross2PedLUD := Cross1PedLUD;
Cross2PedLDU := Cross1PedLUD;
Cross2PedRUD := Cross1PedLUD;
Cross2PedRDU := Cross1PedLUD;

Cross2PedULR := Cross1PedLUD;
Cross2PedURL := Cross1PedLUD;
Cross2PedDLR := Cross1PedLUD;
Cross2PedDRL := Cross1PedLUD;
                      
END_ACTION

ACTION BLINK_YELLOW_SIGNAL:
                        Cross1CarU.GreenLamp := FALSE;
Cross1CarU.YellowLamp := Blinker.OUT;
Cross1CarU.RedLamp := FALSE;

Cross1CarD := Cross1CarU;
Cross1CarL := Cross1CarU;
Cross1CarR := Cross1CarU;

Cross2CarU := Cross1CarU;
Cross2CarD := Cross1CarU;
Cross2CarL := Cross1CarU;
Cross2CarR := Cross1CarU;

Cross1PedLUD.GreenLight := FALSE;
Cross1PedLUD.RedLight := FALSE;
Cross1PedLUD.TimeToSequenceChange := 0;

Cross1PedLDU := Cross1PedLUD;
Cross1PedRUD := Cross1PedLUD;
Cross1PedRDU := Cross1PedLUD;

Cross1PedULR := Cross1PedLUD;
Cross1PedURL := Cross1PedLUD;
Cross1PedDLR := Cross1PedLUD;
Cross1PedDRL := Cross1PedLUD;

Cross2PedLUD := Cross1PedLUD;
Cross2PedLDU := Cross1PedLUD;
Cross2PedRUD := Cross1PedLUD;
Cross2PedRDU := Cross1PedLUD;

Cross2PedULR := Cross1PedLUD;
Cross2PedURL := Cross1PedLUD;
Cross2PedDLR := Cross1PedLUD;
Cross2PedDRL := Cross1PedLUD;
                      
END_ACTION
END_PROGRAM

PROGRAM main
  VAR
    TactTimer : TON;  (* Timer to provide tact for all lights in a synchronized system *)
    vPeriodTime : TIME := TIME#1m2s0ms;  (* Period after the sequence repeats *)
    vElapsedTime : TIME;  (* Elapsed time of the sequence *)
    vTimeToSequenceChange : UDINT;  (* Time in seconds to next sequence change *)
  END_VAR

                    (*Functional description:
This is a program that needs to control two crossroads with cars and pedestrians. The crossroads are one way streets
so cars and pedestrians move in only one direction. It needs to control the traffic lights synchronously
so green wave is kept on the vertical and horizontal lines.
Pedestrian lights work opposite of the car lights so if the vertical line for the cars is green,
the horizontal pedestrians are not allowed to cross and vice versa.
For the pedestrians a time needs to be calculated to show when the green/red light is going to change.

This program implements the sequence diagram given below.
H R   0-30
H Y   28-30 && 60-62
H G   30-60
V R   28-60
V Y   26-28 && 58-60
V G   0-26  && 60-62
P H R 28-60
P H G 0-28
P V R 0-28
P V G 28-60

Simulator decription:
The simulator moves the objects on the road/side walk until they reach a decision point. Decision points
are located next to the related traffic lights. The objects will move only if the traffic light is green
for their direction.
In the simulator the fault monitoring is also active which will stop the objects moving and freeze the lights
so the operator can check where it went wrong. It will also display a message on the screen with the location
and fault reason. During collission or dangerous lights combination all red lights will blink.
To get through the fault situation the operator must enable police control which puts all lights in blinking yellow mode.*)

(*Start the timer and reset it after it expired. Basically count to 85s and then start over*)
TactTimer(IN:=TRUE, PT:=vPeriodTime, ET => vElapsedTime);
IF TactTimer.Q THEN
	TactTimer(IN:=FALSE);
END_IF
(*Calculate next sequence change*)
IF vElapsedTime <= T#28S THEN
	vTimeToSequenceChange := TIME_TO_UDINT(T#28S - vElapsedTime)/1000;
ELSIF vElapsedTime <= T#62S THEN
	vTimeToSequenceChange := TIME_TO_UDINT(T#62S - vElapsedTime)/1000;
END_IF
(* Direction Up, Down traffic light *)
gIO.Cross1CarU.RedLamp    := vElapsedTime >= T#0S  AND vElapsedTime <= T#30S;
gIO.Cross1CarU.YellowLamp := vElapsedTime >= T#28S AND vElapsedTime <= T#30S OR vElapsedTime >= T#60S AND vElapsedTime <= T#62S;
gIO.Cross1CarU.GreenLamp  := vElapsedTime >= T#30S AND vElapsedTime <= T#60S;

(* Mirror the other side of the Up, Down direction *)
gIO.Cross1CarD := gIO.Cross1CarU;
gIO.Cross2CarD := gIO.Cross1CarU;
gIO.Cross2CarU := gIO.Cross1CarU;

(* Direction Left, Right traffic light *)
gIO.Cross1CarL.RedLamp    := vElapsedTime >= T#28S AND vElapsedTime <= T#60S;
gIO.Cross1CarL.YellowLamp := vElapsedTime >= T#26S AND vElapsedTime <= T#28S OR vElapsedTime >= T#58S AND vElapsedTime <= T#60S;
gIO.Cross1CarL.GreenLamp  := vElapsedTime >= T#0S  AND vElapsedTime <= T#26S OR vElapsedTime >= T#60S AND vElapsedTime <= T#62S;

(* Mirror the other side of the Left, Right direction *)
gIO.Cross1CarR := gIO.Cross1CarL;
gIO.Cross2CarR := gIO.Cross1CarL;
gIO.Cross2CarL := gIO.Cross1CarL;

(*Pedestrians*)
(*If left <-> right cars are going. Up <-> down pedestrians stop. Else go*)
IF gIO.Cross1CarL.GreenLamp OR gIO.Cross1CarL.YellowLamp  THEN
	gIO.Cross1PedLDU.RedLight := TRUE;
	gIO.Cross1PedLDU.GreenLight := FALSE;
	
ELSIF gIO.Cross1CarL.RedLamp THEN
	gIO.Cross1PedLDU.RedLight := FALSE;
	gIO.Cross1PedLDU.GreenLight := TRUE;

END_IF
gIO.Cross1PedLDU.TimeToSequenceChange := UDINT_TO_UINT(vTimeToSequenceChange);

(*Just copy all of the up and downs as they behave the same*)
gIO.Cross1PedLUD := gIO.Cross1PedLDU;
gIO.Cross1PedRUD := gIO.Cross1PedLDU;
gIO.Cross1PedRDU := gIO.Cross1PedLDU;
gIO.Cross2PedLDU := gIO.Cross1PedLDU;
gIO.Cross2PedLUD := gIO.Cross1PedLDU;
gIO.Cross2PedRUD := gIO.Cross1PedLDU;
gIO.Cross2PedRDU := gIO.Cross1PedLDU;

(*If up <-> Down cars are going. Left <-> right pedestrians stop. Else go*)
IF gIO.Cross1CarU.GreenLamp OR gIO.Cross1CarU.YellowLamp THEN
	gIO.Cross1PedULR.RedLight := TRUE;
	gIO.Cross1PedULR.GreenLight := FALSE;

ELSIF gIO.Cross1CarU.RedLamp THEN
	gIO.Cross1PedULR.RedLight := FALSE;
	gIO.Cross1PedULR.GreenLight := TRUE;
END_IF
gIO.Cross1PedULR.TimeToSequenceChange := UDINT_TO_UINT(vTimeToSequenceChange);

(*Just copy all of the lefts and rights as they behave the same*)
gIO.Cross1PedURL := gIO.Cross1PedULR;
gIO.Cross1PedDLR := gIO.Cross1PedULR;
gIO.Cross1PedDRL := gIO.Cross1PedULR;
gIO.Cross2PedULR := gIO.Cross1PedULR;
gIO.Cross2PedURL := gIO.Cross1PedULR;
gIO.Cross2PedDLR := gIO.Cross1PedULR;
gIO.Cross2PedDRL := gIO.Cross1PedULR;
                  
END_PROGRAM

CONFIGURATION SoftPLC
  RESOURCE Application ON PLC
    {attribute 'qualified_only'}
    VAR_GLOBAL  (* gIO *)
      Cross1CarU : trafficLightCars;  (* Car traffic light DO - Crossroad 1 - Cars going up to down *)
      Cross1CarD : trafficLightCars;  (* Car traffic light DO - Crossroad 1 - Cars going down to up *)
      Cross1CarL : trafficLightCars;  (* Car traffic light DO - Crossroad 1 - Cars going left to right *)
      Cross1CarR : trafficLightCars;  (* Car traffic light DO - Crossroad 1 - Cars going right to left *)
      Cross2CarU : trafficLightCars;  (* Car traffic light DO - Crossroad 2 - Cars going up to down *)
      Cross2CarD : trafficLightCars;  (* Car traffic light DO - Crossroad 2 - Cars going down to up *)
      Cross2CarL : trafficLightCars;  (* Car traffic light DO - Crossroad 2 - Cars going left to right *)
      Cross2CarR : trafficLightCars;  (* Car traffic light DO - Crossroad 2 - Cars going right to left *)
      Cross1PedLUD : trafficLightPed;  (* Pedestrian light DO - Crossroad 1 - Pedestrians going up to down on left side *)
      Cross1PedLDU : trafficLightPed;  (* Pedestrian light DO - Crossroad 1 - Pedestrians going down to up on left side *)
      Cross1PedRUD : trafficLightPed;  (* Pedestrian light DO - Crossroad 1 - Pedestrians going up to down on right side *)
      Cross1PedRDU : trafficLightPed;  (* Pedestrian light DO - Crossroad 1 - Pedestrians going down to up on right side *)
      Cross1PedULR : trafficLightPed;  (* Pedestrian light DO - Crossroad 1 - Pedestrians going left to right on upper side *)
      Cross1PedURL : trafficLightPed;  (* Pedestrian light DO - Crossroad 1 - Pedestrians going right to left on upper side *)
      Cross1PedDLR : trafficLightPed;  (* Pedestrian light DO - Crossroad 1 - Pedestrians going left to right on lower side *)
      Cross1PedDRL : trafficLightPed;  (* Pedestrian light DO - Crossroad 1 - Pedestrians going right to left on lower side *)
      Cross2PedLUD : trafficLightPed;  (* Pedestrian light DO - Crossroad 2 - Pedestrians going up to down on left side *)
      Cross2PedLDU : trafficLightPed;  (* Pedestrian light DO - Crossroad 2 - Pedestrians going down to up on left side *)
      Cross2PedRUD : trafficLightPed;  (* Pedestrian light DO - Crossroad 2 - Pedestrians going up to down on right side *)
      Cross2PedRDU : trafficLightPed;  (* Pedestrian light DO - Crossroad 2 - Pedestrians going down to up on right side *)
      Cross2PedULR : trafficLightPed;  (* Pedestrian light DO - Crossroad 2 - Pedestrians going left to right on upper side *)
      Cross2PedURL : trafficLightPed;  (* Pedestrian light DO - Crossroad 2 - Pedestrians going right to left on upper side *)
      Cross2PedDLR : trafficLightPed;  (* Pedestrian light DO - Crossroad 2 - Pedestrians going left to right on lower side *)
      Cross2PedDRL : trafficLightPed;  (* Pedestrian light DO - Crossroad 2 - Pedestrians going right to left on lower side *)
      PoliceModeActivated : BOOL;  (* DI Police mode is activated *)
    END_VAR
    TASK VISU_TASK(INTERVAL := T#50ms, PRIORITY := 31);
    TASK Task(INTERVAL := T#5ms, PRIORITY := 1);
    PROGRAM VisuElems.Visu_Prg WITH VISU_TASK : VisuElems.Visu_Prg;
    PROGRAM main WITH Task : main;
    PROGRAM simulator WITH Task : simulator;
  END_RESOURCE
END_CONFIGURATION
